PROGRAM Q3
VAR
	S1 : BOOL := FALSE; // First Switch
	S2 : BOOL := FALSE; // Second Switch
	M1 : BOOL := FALSE; // Motor
END_VAR

// To run:
// Paste the following into the MAIN file
// Q3();

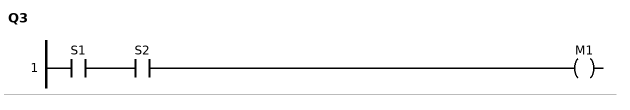
// NETWORK 1
M1 := S1 AND S2;

END_PROGRAM

(* stored: Version 1.1.0.1, ProductVersion 3.1.4024.12
   POU Q3: Id {c48f14dc-a332-42f7-943a-4fde817c8093}, SpecialFunc None *)
